TYPE TcoTixonPickVibroBasic_Config_v_1_x_x EXTENDS TcoTixonGenericPickConfig : STRUCT
    {attribute addProperty Name "<#Error time separator #> - T_SEP_ERROR"}
    ErrorTimeSeparator : TIME := T#0S;
    {attribute addProperty Name "<#Error time buffer #> - T_BUFF_ERROR"}
    ErrorTimeBuffer : TIME := T#0S;
    {attribute addProperty Name "<#Error time Hopper #> - T_HOP_ERROR"}
    ErrorTimeHopper : TIME := T#0S;
END_STRUCT
END_TYPE

(* stored: Version 1.1.0.1, ProductVersion 3.1.4024.12
   DUT TcoTixonPickVibroBasic_Config_v_1_x_x: Id {331d5491-a789-0dbb-1ee3-d9aaf078a9f6} *)
